DATA_BLOCK "dbArchiveControlExhaust"
{ S7_Optimized_Access := 'TRUE' }
VERSION : 0.8
NON_RETAIN
"fbArchiveControlExhaust"

BEGIN

END_DATA_BLOCK

